(* CoDeSys 2.3 export: MNG_DATAARRAY.EXP *)

(* Data type in MNG_TCPIP *)
TYPE MNG_DataArray : ARRAY[1..MNG_BUFFER_SIZE] OF DWORD; (* user data of max. length *)
END_TYPE
